// Mitsubishi GX Works2 project: PLC-GROUP21   PLC: FX3G

// global labels: Global1
VAR_GLOBAL
  end_day AT M10 : BOOL;
END_VAR
VAR_GLOBAL CONSTANT
  constant_0 : REAL;
END_VAR
VAR_GLOBAL
  oat_quantity AT D1100 : REAL;
  protein_quantity AT D1150 : REAL;
  honey_quantity AT D1200 : REAL;
  Total_prodact AT D1250 : REAL;
  oat_input AT D1100 : REAL;
  protein_input AT D1150 : REAL;
  honey_input AT D1200 : REAL;
END_VAR
VAR_GLOBAL CONSTANT
  constant_400 : REAL := 400;
  constant_320 : REAL := 320;
  constant_160 : REAL := 160;
END_VAR
VAR_GLOBAL
  check_quantity AT M50 : BOOL;
  start_day_button AT X007 : BOOL;
  not_end AT Y000 : BOOL;
  Analoginput1 AT D8280 : INT;
  bar_type AT D1300 : REAL;
  normalized_input AT M60 : BOOL;
END_VAR
VAR_GLOBAL CONSTANT
  constant_5 : REAL := 5;
END_VAR
VAR_GLOBAL
  classic AT M65 : BOOL;
END_VAR
VAR_GLOBAL CONSTANT
  constant_10 : REAL := 10;
END_VAR
VAR_GLOBAL
  protein AT M70 : BOOL;
  start_mixing_procedure AT X003 : BOOL;
  mixing_in_progress AT Y003 : BOOL;
  help_blink AT M105 : BOOL;
  TC_1 AT TC1 : BOOL;
END_VAR
VAR_GLOBAL CONSTANT
  constant_40 : REAL := 40;
END_VAR
VAR_GLOBAL
  stop_blinking_y1 AT TS1 : BOOL;
  blink_y1 AT Y001 : BOOL;
  stop_blinking_y2 AT TS2 : BOOL;
  TC_2 AT TC2 : BOOL;
  blink_y2 AT Y002 : BOOL;
END_VAR
VAR_GLOBAL CONSTANT
  constant_50 : INT := 50;
END_VAR
VAR_GLOBAL
  TC_5 AT TC5 : BOOL;
  start_packaging AT X006 : BOOL;
  package_one_bar AT X000 : BOOL;
  emergency_button AT X005 : BOOL;
  mix_tank AT D1400 : REAL;
END_VAR
VAR_GLOBAL CONSTANT
  constant_120 : REAL := 120;
  constant_240 : REAL := 240;
END_VAR
VAR_GLOBAL
  start_baking_process AT X002 : BOOL;
  oven AT D1450 : REAL;
END_VAR
VAR_GLOBAL CONSTANT
  constant_8 : INT := 8;
END_VAR
VAR_GLOBAL
  packaging_light AT Y004 : BOOL;
END_VAR
VAR_GLOBAL CONSTANT
  constant_1 : INT := 1;
END_VAR
VAR_GLOBAL
  Analog_output AT D8282 : INT;
END_VAR
VAR_GLOBAL CONSTANT
  const_40 : INT := 40;
END_VAR
VAR_GLOBAL
  TC_8 AT TC8 : BOOL;
END_VAR
VAR_GLOBAL CONSTANT
  const_10 : INT := 10;
END_VAR
VAR_GLOBAL
  TC_9 AT TC9 : BOOL;
  Timer_second AT TS9 : BOOL;
  Timer_first AT TS8 : BOOL;
  count_first_bar AT CC1 : BOOL;
  count_7_more_bars AT CC2 : BOOL;
  package_one_bar_out AT CS1 : BOOL;
  count_7_bars_out AT CS2 : BOOL;
END_VAR
VAR_GLOBAL CONSTANT
  const_1 : REAL := 1;
END_VAR
VAR_GLOBAL
  cant_produce AT M75 : BOOL;
END_VAR
VAR_GLOBAL CONSTANT
  const_0 : INT;
END_VAR
VAR_GLOBAL
  move_quantity AT M170 : BOOL;
  help_y3 AT TS5 : BOOL;
END_VAR

// task Task_01 (event TRUE, interval 0, priority 31): POU_01

PROGRAM POU_01
(* structured ladder/FBD written out as ST: instructions are called as NAME(EN, inputs, outputs); _pN, _eN, _tN stand for wires *)
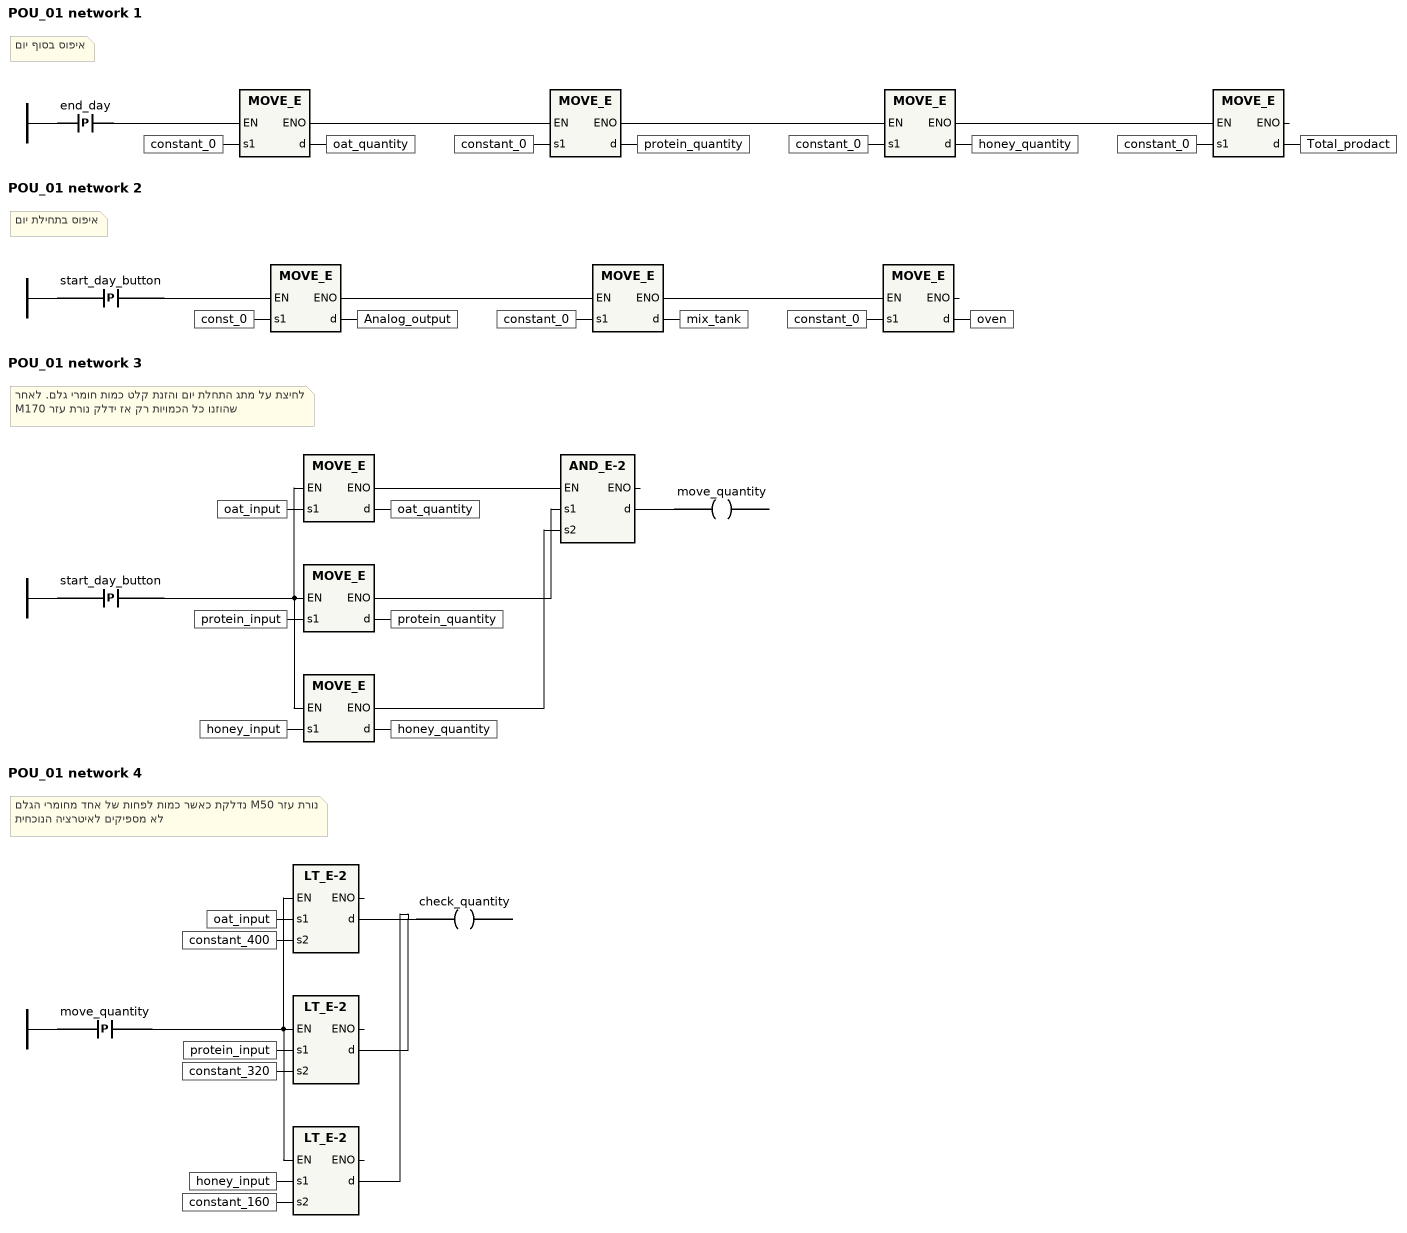
(* network 1 *)
(* איפוס בסוף יום *)
_e1 := MOVE_E(LDP(TRUE, end_day), constant_0, oat_quantity);
_e2 := MOVE_E(_e1, constant_0, protein_quantity);
_e3 := MOVE_E(_e2, constant_0, honey_quantity);
MOVE_E(_e3, constant_0, Total_prodact);
(* network 2 *)
(* איפוס בתחילת יום *)
_e1 := MOVE_E(LDP(TRUE, start_day_button), const_0, Analog_output);
_e2 := MOVE_E(_e1, constant_0, mix_tank);
MOVE_E(_e2, constant_0, oven);
(* network 3 *)
(* לחיצת על מתג התחלת יום והזנת קלט כמות חומרי גלם. לאחר שהוזנו כל הכמויות רק אז ידלק נורת עזר M170 *)
_p1 := LDP(TRUE, start_day_button);
_e2 := MOVE_E(_p1, oat_input, oat_quantity);
_e3 := MOVE_E(_p1, protein_input, protein_quantity);
_e4 := MOVE_E(_p1, honey_input, honey_quantity);
AND_E(_e2, _e3, _e4, _t5);
move_quantity := _t5;
(* network 4 *)
(* נורת עזר M50 נדלקת כאשר כמות לפחות של אחד מחומרי הגלם לא מספיקים לאיטרציה הנוכחית *)
_p1 := LDP(TRUE, move_quantity);
LT_E(_p1, oat_input, constant_400, _t2);
LT_E(_p1, protein_input, constant_320, _t3);
LT_E(_p1, honey_input, constant_160, _t4);
check_quantity := _t2 OR _t3 OR _t4;
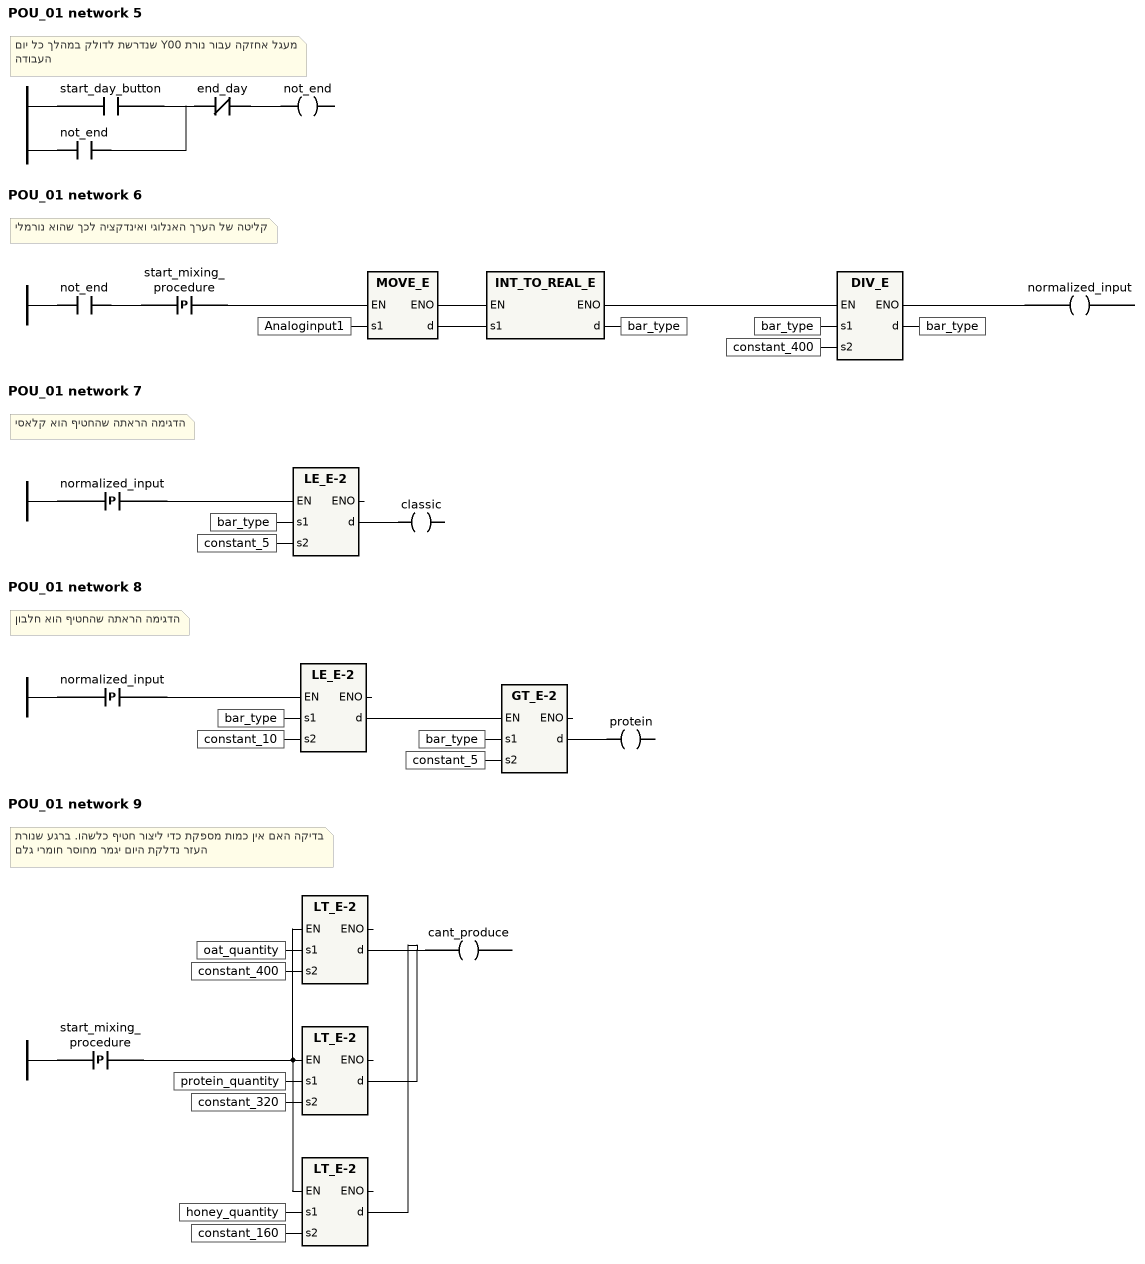
(* network 5 *)
(* מעגל אחזקה עבור נורת Y00 שנדרשת לדולק במהלך כל יום העבודה *)
not_end := (start_day_button OR not_end) AND NOT end_day;
(* network 6 *)
(* קליטה של הערך האנלוגי ואינדקציה לכך שהוא נורמלי *)
_e2 := MOVE_E(not_end AND LDP(TRUE, start_mixing_procedure), Analoginput1, _t1);
_e3 := INT_TO_REAL_E(_e2, _t1, bar_type);
_e4 := DIV_E(_e3, bar_type, constant_400, bar_type);
normalized_input := _e4;
(* network 7 *)
(* הדגימה הראתה שהחטיף הוא קלאסי *)
LE_E(LDP(TRUE, normalized_input), bar_type, constant_5, _t1);
classic := _t1;
(* network 8 *)
(* הדגימה הראתה שהחטיף הוא חלבון *)
LE_E(LDP(TRUE, normalized_input), bar_type, constant_10, _t1);
GT_E(_t1, bar_type, constant_5, _t2);
protein := _t2;
(* network 9 *)
(* בדיקה האם אין כמות מספקת כדי ליצור חטיף כלשהו. ברגע שנורת העזר נדלקת היום יגמר מחוסר חומרי גלם *)
_p1 := LDP(TRUE, start_mixing_procedure);
LT_E(_p1, oat_quantity, constant_400, _t2);
LT_E(_p1, protein_quantity, constant_320, _t3);
LT_E(_p1, honey_quantity, constant_160, _t4);
cant_produce := _t2 OR _t3 OR _t4;
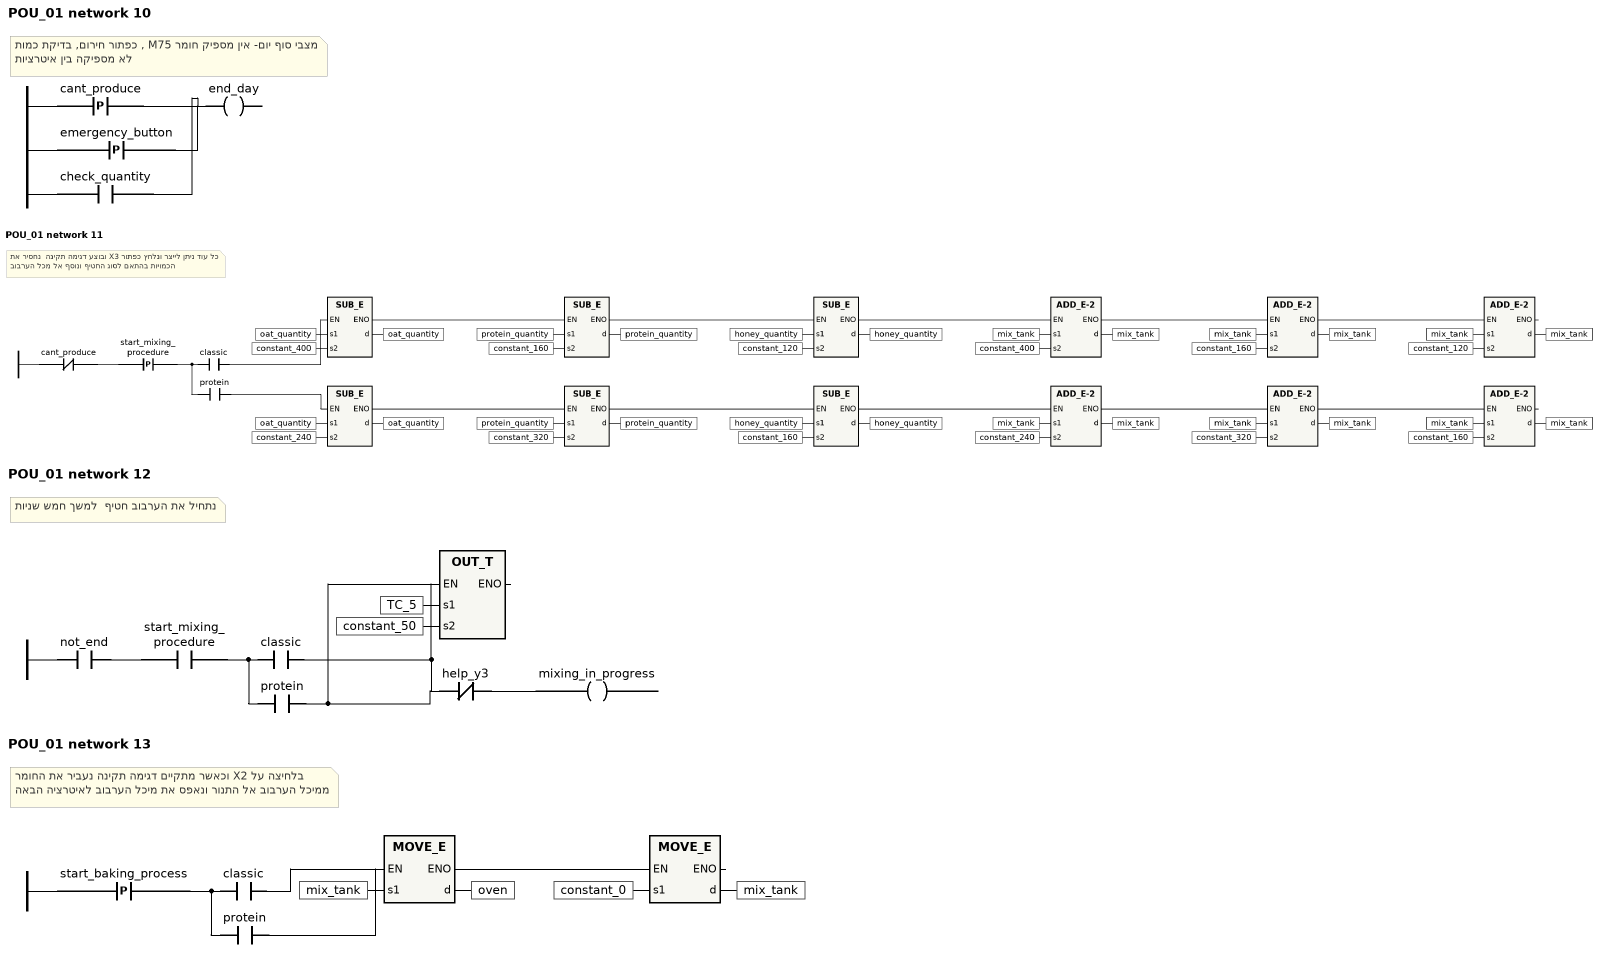
(* network 10 *)
(* מצבי סוף יום- אין מספיק חומר M75 , כפתור חירום, בדיקת כמות לא מספיקה בין איטרציות *)
end_day := LDP(TRUE, cant_produce) OR LDP(TRUE, emergency_button) OR check_quantity;
(* network 11 *)
(* כל עוד ניתן לייצר ונלחץ כפתור X3 ובוצע דגימה תקינה  נחסיר את הכמויות בהתאם לסוג החטיף ונוסף אל מכל הערבוב *)
_p1 := NOT cant_produce AND LDP(TRUE, start_mixing_procedure);
_e2 := SUB_E(_p1 AND classic, oat_quantity, constant_400, oat_quantity);
_e3 := SUB_E(_e2, protein_quantity, constant_160, protein_quantity);
_e4 := SUB_E(_e3, honey_quantity, constant_120, honey_quantity);
_e5 := ADD_E(_e4, mix_tank, constant_400, mix_tank);
_e6 := ADD_E(_e5, mix_tank, constant_160, mix_tank);
ADD_E(_e6, mix_tank, constant_120, mix_tank);
_e7 := SUB_E(_p1 AND protein, oat_quantity, constant_240, oat_quantity);
_e8 := SUB_E(_e7, protein_quantity, constant_320, protein_quantity);
_e9 := SUB_E(_e8, honey_quantity, constant_160, honey_quantity);
_e10 := ADD_E(_e9, mix_tank, constant_240, mix_tank);
_e11 := ADD_E(_e10, mix_tank, constant_320, mix_tank);
ADD_E(_e11, mix_tank, constant_160, mix_tank);
(* network 12 *)
(* נתחיל את הערבוב חטיף  למשך חמש שניות *)
_p1 := not_end AND start_mixing_procedure;
_p2 := (_p1 AND classic) OR (_p1 AND protein);
OUT_T(_p2, TC_5, constant_50);
mixing_in_progress := _p2 AND NOT help_y3;
(* network 13 *)
(* בלחיצה על X2 וכאשר מתקיים דגימה תקינה נעביר את החומר ממיכל הערבוב אל התנור ונאפס את מיכל הערבוב לאיטרציה הבאה *)
_p1 := LDP(TRUE, start_baking_process);
_e2 := MOVE_E((_p1 AND classic) OR (_p1 AND protein), mix_tank, oven);
MOVE_E(_e2, constant_0, mix_tank);
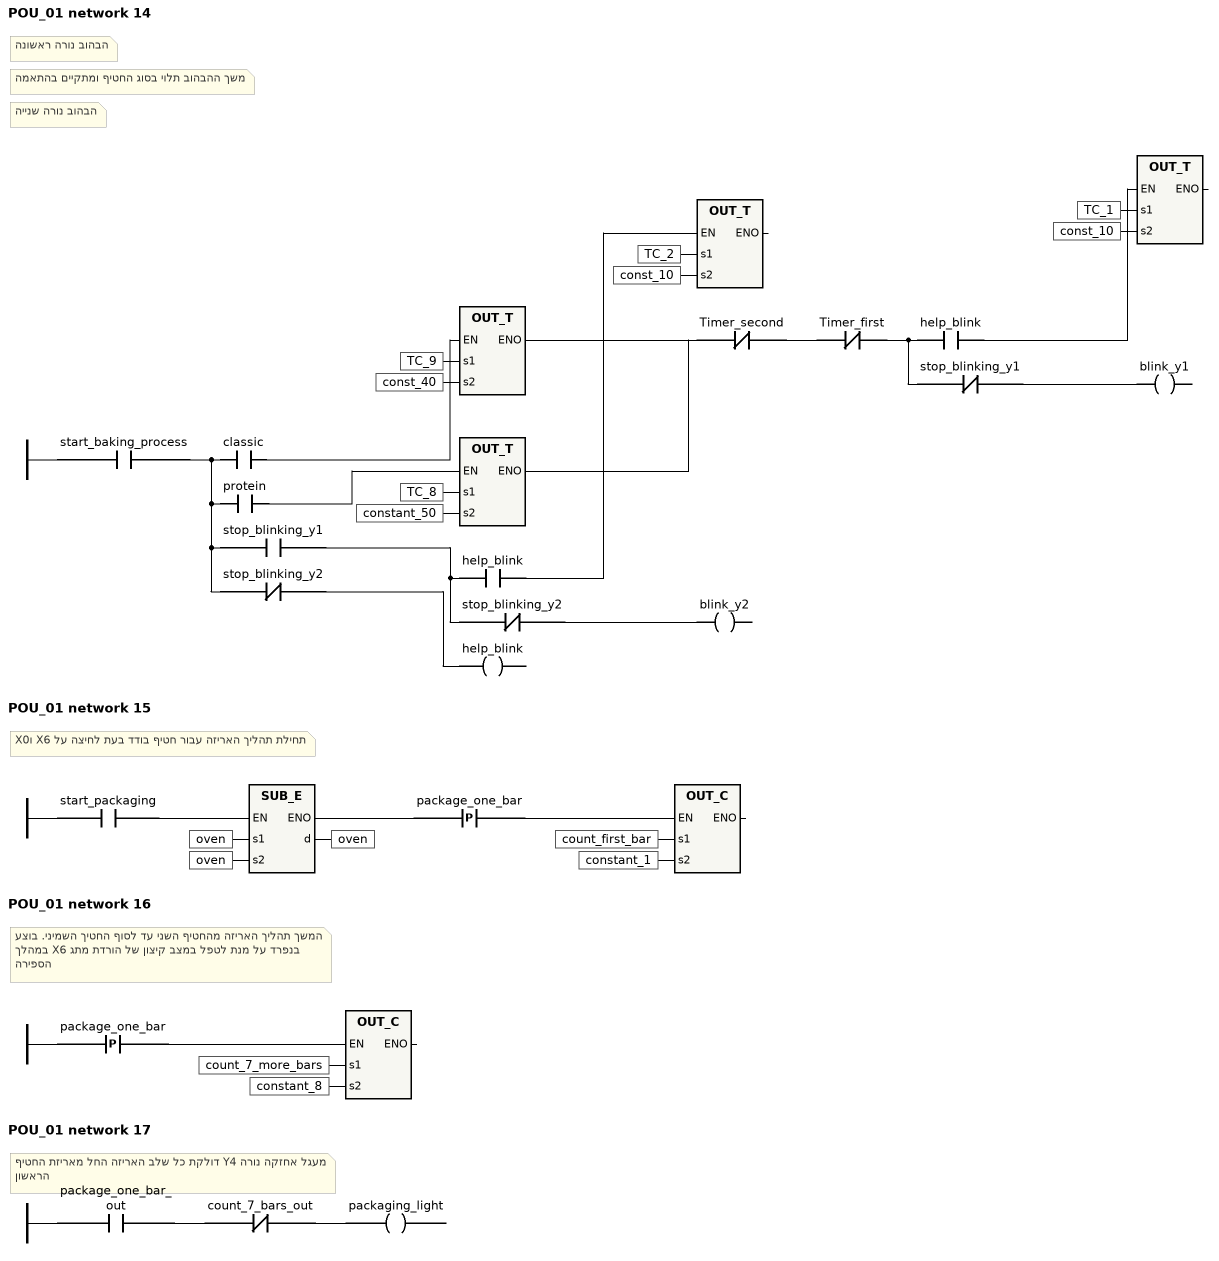
(* network 14 *)
(* הבהוב נורה ראשונה *)
(* משך ההבהוב תלוי בסוג החטיף ומתקיים בהתאמה *)
(* הבהוב נורה שנייה *)
_e1 := OUT_T(start_baking_process AND classic, TC_9, const_40);
_e2 := OUT_T(start_baking_process AND protein, TC_8, constant_50);
_p3 := ((_e1 OR _e2) AND NOT Timer_second) AND NOT Timer_first;
OUT_T(_p3 AND help_blink, TC_1, const_10);
blink_y1 := _p3 AND NOT stop_blinking_y1;
_p4 := start_baking_process AND stop_blinking_y1;
OUT_T(_p4 AND help_blink, TC_2, const_10);
blink_y2 := _p4 AND NOT stop_blinking_y2;
help_blink := start_baking_process AND NOT stop_blinking_y2;
(* network 15 *)
(* תחילת תהליך האריזה עבור חטיף בודד בעת לחיצה על X6 וX0 *)
_e1 := SUB_E(start_packaging, oven, oven, oven);
OUT_C(_e1 AND LDP(TRUE, package_one_bar), count_first_bar, constant_1);
(* network 16 *)
(* המשך תהליך האריזה מהחטיף השני עד לסוף החטיך השמיני. בוצע בנפרד על מנת לטפל במצב קיצון של הורדת מתג X6 במהלך הספירה *)
OUT_C(LDP(TRUE, package_one_bar), count_7_more_bars, constant_8);
(* network 17 *)
(* מעגל אחזקה נורה Y4 דולקת כל שלב האריזה החל מאריזת החטיף הראשון *)
packaging_light := package_one_bar_out AND NOT count_7_bars_out;
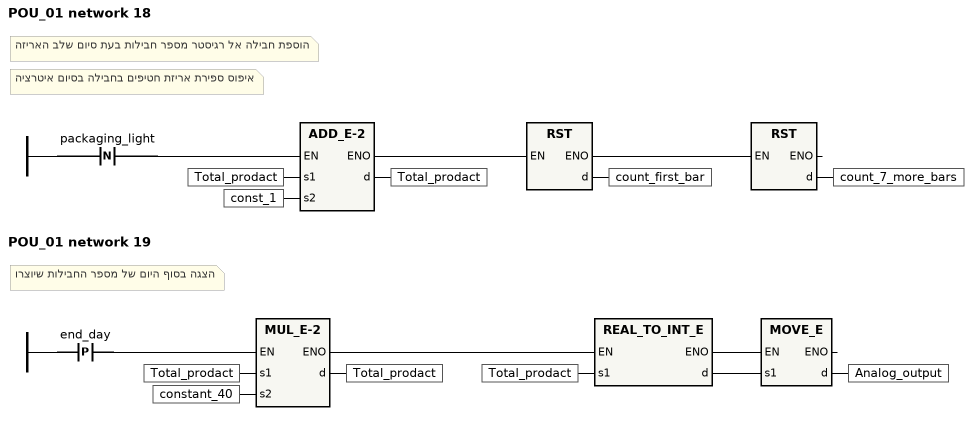
(* network 18 *)
(* הוספת חבילה אל רגיסטר מספר חבילות בעת סיום שלב האריזה *)
(* איפוס ספירת אריזת חטיפים בחבילה בסיום איטרציה *)
_e1 := ADD_E(LDF(TRUE, packaging_light), Total_prodact, const_1, Total_prodact);
_e2 := RST(_e1, count_first_bar);
RST(_e2, count_7_more_bars);
(* network 19 *)
(* הצגה בסוף היום של מספר החבילות שיוצרו *)
_e1 := MUL_E(LDP(TRUE, end_day), Total_prodact, constant_40, Total_prodact);
_e3 := REAL_TO_INT_E(_e1, Total_prodact, _t2);
MOVE_E(_e3, _t2, Analog_output);
END_PROGRAM
